{attribute 'qualified_only'}
{attribute 'strict'}
TYPE Sensies :
(
	Sick := 0,
	Pilz := 1,
	Parker := 2,
	Bosh := 3
)USINT;
END_TYPE

(* stored: Version 1.1.0.1, ProductVersion 3.1.4024.12
   DUT Sensies: Id {837b9654-2b4a-40b1-813f-0431aaa6e7fc} *)
